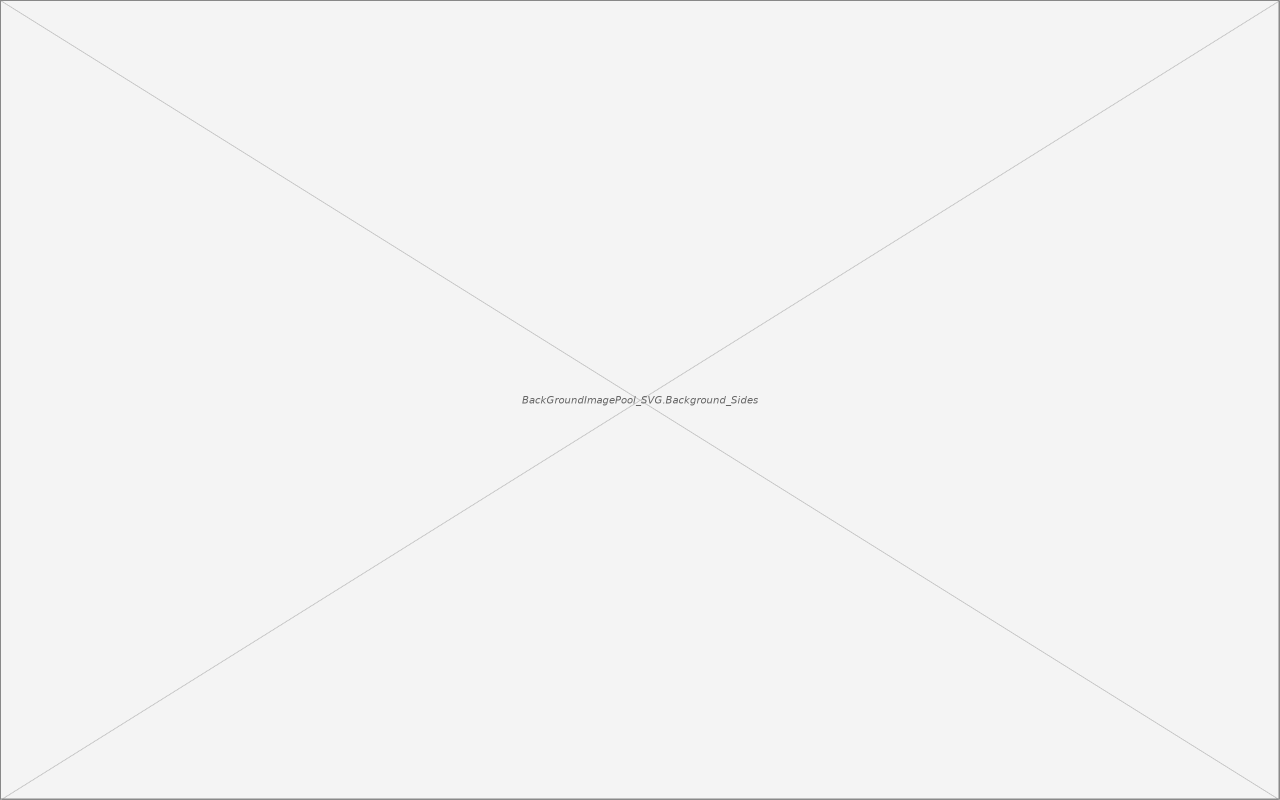
VISUALIZATION BG_Borders  // 1280x800
    Image (0,710 1280x90), image: BackGroundImagePool_SVG.Background_Bottom
    Image (0,0 1280x800), image: BackGroundImagePool_SVG.Background_Sides
END_VISUALIZATION

(* stored: Version 1.1.0.1, ProductVersion 3.1.4024.11
   Visu BG_Borders: Id {7601f2db-9dda-4b85-a89f-5559794de405} *)
